// TIA Portal V16 export
// export: Created 2023-08-28T09:37:51.3805988Z, ExportSetting WithDefaults, DisplayName Totally Integrated Automation Portal, DisplayVersion V16 Update 6, DisplayName TIA Portal Version Control Interface, DisplayVersion V16 Update 2, DisplayName TIA Portal Openness, DisplayVersion V16 Update 6, DisplayName STEP 7 Professional, DisplayVersion V16 Update 6, DisplayName STEP 7 Safety, DisplayVersion V16, DisplayName WinCC Advanced, DisplayVersion V16 Update 6
DATA_BLOCK "dbMasterData"   // DB35
{ S7_Optimized_Access := 'FALSE' }
VERSION : 0.1
// stored: AutoNumber false, DBAccessibleFromOPCUA true, IsOnlyStoredInLoadMemory false, IsWriteProtectedInAS false
   VAR
      ID6_aktualny_przeływu_Adres_33057 { S7_SetPoint := 'True'} : "typeDataABB_real";   // wielkość przepływu / Wartość aktualnego przepływu
      ID6_Licznik_suma_VF_Adres_33063 : "typeDataABB_real";   // licznik objętości VF / Stan licznika objętości dla przepływu w przód VF
      ID6_Licznik_suma_VR_Adres_33065 { S7_SetPoint := 'True'} : "typeDataABB_real";   // licznik objętości VR / Stan licznika objętości dla przepływu w tył VR
      ID6__VD_Adres_6 { S7_SetPoint := 'True'} : "typeDataABB_real";   // Stan bieżącego różnicowego licznika objętości VD
      ID6___GF_Adres_8 { S7_SetPoint := 'True'} : "typeDataABB_real";   // Stan głównego licznika objętości dla przepływu w przód GF
      ID6__GR_Adres_10 { S7_SetPoint := 'True'} : "typeDataABB_real";   // Sta ngłownego licznika objętości dla przepływu w tył GR
      ID6__GD_Adres_12 { S7_SetPoint := 'True'} : "typeDataABB_real";   // Stan głownego licznika różnicowego GD
      ID6__1000 { S7_SetPoint := 'True'} : "typeDataInverter_Word";   // 8-przekrodzony zakres pracy przetwornika, 20-otwarty obwód cewki, 21zwarcie w obwodzie cewki, 26-brak cieczy w czujniku
      data_rez_Wielkość_przeływu_Adres_0 { S7_SetPoint := 'True'} : "typeDataABB_real";   // wielkość przepływu / Wartość aktualnego przepływu
      data_rez_Licznik_objętość_VF_Adres_2 { S7_SetPoint := 'True'} : "typeDataABB_real";   // licznik objętości VF / Stan licznika objętości dla przepływu w przód VF
      data_rez_Licznik_objętość_VR_Adres_4 { S7_SetPoint := 'True'} : "typeDataABB_real";   // licznik objętości VR / Stan licznika objętości dla przepływu w tył VR
      data_rez_Licznik_różnicowy_VD_Adres_6 { S7_SetPoint := 'True'} : "typeDataABB_real";   // licznik różnicy / Stan bieżącego różnicowego licznika objętości VD
      data_rez_Stan_licz_bjętości_GF_Adres_8 { S7_SetPoint := 'True'} : "typeDataABB_real";   // licznik objetosci GF / Stan głównego licznika objętości dla przepływu w przód GF
      data_rez_Stan_licz_bjętości_GR_Adres_10 { S7_SetPoint := 'True'} : "typeDataABB_real";   // licznik objetości GR / Sta ngłownego licznika objętości dla przepływu w tył GR
      data_rez_Stan_licz_rózicowego_obj_GD_Adres_12 { S7_SetPoint := 'True'} : "typeDataABB_real";   // licznik róznicowy / Stan głownego licznika różnicowego GD
      data_rez_Stan_urządzenia_1000 { S7_SetPoint := 'True'} : "typeDataInverter_Word";   // stan urządzenia / 8-przekrodzony zakres pracy przetwornika, 20-otwarty obwód cewki, 21zwarcie w obwodzie cewki, 26-brak cieczy w czujniku
      ID26_Inver_Control_word_416000_Fal { S7_SetPoint := 'True'} : "typeDataInverter_Word";   // Sowo komtrolneCTW falownika [Uint16, index 0]
      ID26_Inver_setpoint_ref_416020_Fal { S7_SetPoint := 'True'} : "typeDataInverter_Word";   // Słowo wartość zadana Hz [Int16, index -1]
      ID26_Inver_Status_word_416030_Fal { S7_SetPoint := 'True'} : "typeDataInverter_Word";   // Słowo statusu STW falownika [Uint16, index 0]
      ID26_Inver_Frequency_416130_Fal { S7_SetPoint := 'True'} : "typeDataInverter_Word";   // Słowo częstotliwość na wyjściu [Uint16, index -1]
      ID26_Inver_MotorCurrent_416140_Fal { S7_SetPoint := 'True'} : "typeDataInverter_Word";   // Słowo częstotliwość na wyjściu [Uint16, index -2]
      ID26_Inver_DC_Voltage_416300_Fal { S7_SetPoint := 'True'} : "typeDataInverter_Word";   // Słowo napięcia DC na szynie [Uint16, index 0]
      ID26_Inver_Temp_416340_Fal { S7_SetPoint := 'True'} : "typeDataInverter_Word";   // Słowo temperatura invertera [Uint8, index 0]
      ID26_Inver_NomCurrent_416360_Fal { S7_SetPoint := 'True'} : "typeDataInverter_Word";   // Słowo nominalna wartośc prądu falonika[Uint16, index -2]
      ID26_Inver_MaxCurrent_416370_Fal { S7_SetPoint := 'True'} : "typeDataInverter_Word";   // Słowo max prąd falownika [Uint16, index -2]
      ID26_Inver_InDigit_416600_Fal { S7_SetPoint := 'True'} : "typeDataInverter_Word";   // Słowo mampa wejść 18,19,27,33 [Uint16, index -0]
      ID26_Inver_HourWork_415010_Fal { S7_SetPoint := 'True'} : "typeDataInverter_DWord";   // Podwójne słowo czasu pracy falownika [Int32, index -0]
      ID26_Inver_OverTemp_415040_Fal { S7_SetPoint := 'True'} : "typeDataInverter_Word";   // Sowo statusu przekroczenie temperatury[Uint16, index 0]
      ID26_Inver_OverVolts_415050_Fal { S7_SetPoint := 'True'} : "typeDataInverter_Word";   // Sowo statusu przekroczenie napięcia[Uint16, index 0]
      data_RTU_value_0 { S7_SetPoint := 'True'} : "typeDataABB_real";   // Wartość 0.0 pomocnicza wyświetlana podczas błędu pomiaru
   END_VAR
BEGIN
   data_RTU_value_0.data[0] := 0.0;
END_DATA_BLOCK
